// Mitsubishi GX Works2 project: 240430_timechart03_자기유지gxw   PLC: Q03UDV

PROGRAM MAIN
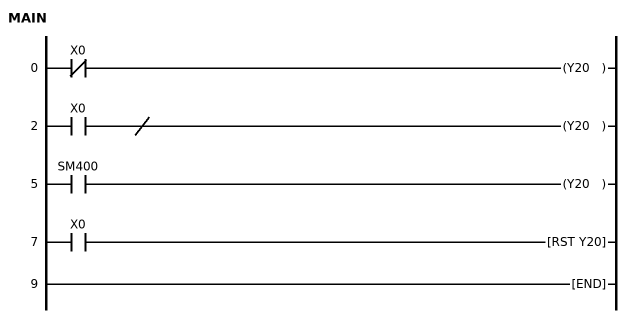
0     LDI     X0
      OUT     Y20
2     LD      X0
      INV
      OUT     Y20
5     LD      SM400
      OUT     Y20
7     LD      X0
      RST     Y20
9     END
END_PROGRAM
